Universal Robots PolyScope program: pallet_126.urp

Program pallet_126 (createdIn=3.2.19293 lastSavedIn=3.2.19293 directory=/programs installation=default robotSerialNumber=2015351391)
Calibrated DH parameters: a=[0.000352, -0.161198, -0.373486, 0.00005, 0.000049, 0]; d=[0.089268, 352.477598, -320.08558, -32.281492, 0.094939, 0.082518]; alpha=[1.570728, 0.001116, -0.003686, 1.571189, -1.570572, 0]; deltaTheta=[-0.000012, 1.181849, -1.491165, 0.309495, -0.000007, 0.000025]
Robot Program (runOnlyOnce=false motionType=MoveJ speed=1.047198 acceleration=1.396263 recalculateMotions=false)
  Pallet pattern(dimensionality=Square firstAxisCount=3 secondAxisCount=3 thirdAxisCount=5 motionType=MoveL speed=0.25 acceleration=1.2 recalculateMotions=false, counterVariable(name=cnt_1, initializeExpression=0), patternPoseVariable(name=位姿_1), feature=Base, children(Waypoint(type=Fixed name=a1st_Corner_1, position(joints=2.5763556957244873, -2.0812442938434046, -2.0229433218585413, -0.5034664312945765, 1.591776967048645, -0.26194888750185186 pose=-0.39287493474301816, 0.3789089223527664, 0.06616154798695834, -2.460791536512403, -1.8027009363597946, 0.090316902258006), poseInFeatureCoordinates=[-0.392875, 0.378909, 0.066162, -2.460792, -1.802701, 0.090317], outputFlangePose=[-0.392865, 0.378909, 0.066161, -2.460798, -1.802654, 0.090216]), Waypoint(type=Fixed name=a2nd_Corner_1, position(joints=2.3224451541900635, -2.320186440144674, -1.5487983862506312, -0.7482627073871058, 1.5784262418746948, -0.5291169325457972 pose=-0.386611770730188, 0.5758943302513561, 0.06650521658612327, -2.446947628948111, -1.8165459438339622, 0.030894912998256457), poseInFeatureCoordinates=[-0.386612, 0.575894, 0.066505, -2.446948, -1.816546, 0.030895], outputFlangePose=[-0.386628, 0.575892, 0.066482, -2.446977, -1.816542, 0.030841]), Waypoint(type=Fixed name=a3rd_Corner_1, position(joints=2.0719354207892664, -2.1626037568261713, -1.8315477023713154, -0.6285018266102558, 1.6020367779501523, -0.7786933796104183 pose=-0.19145307853450216, 0.5759079217417217, 0.07306667136931888, -2.446955511533883, -1.8165637951887514, 0.030572269090385032), poseInFeatureCoordinates=[-0.191453, 0.575908, 0.073067, -2.446956, -1.816564, 0.030572], outputFlangePose=[-0.191468, 0.575892, 0.07306, -2.446977, -1.816542, 0.030841]), Waypoint(type=Fixed name=a4th_Corner_1, position(joints=2.3161087418842667, -1.8639255502475685, -2.380638872250877, -0.3727480295157033, 1.579937380718258, -0.5354962677601893 pose=-0.19147099564377815, 0.37025084098707506, 0.07306665267587242, -2.4469490165306196, -1.8165403427476172, 0.03091275584599603), poseInFeatureCoordinates=[-0.191471, 0.370251, 0.073067, -2.446949, -1.81654, 0.030913], outputFlangePose=[-0.191468, 0.370234, 0.07306, -2.446977, -1.816542, 0.030841]))); actionSequence(name=托盘序列 motionType=MoveL speed=0.25 acceleration=1.2 recalculateMotions=false, anchorWaypoint(type=Fixed name=模式点_1, position(joints=2.5763556957244873, -2.0812442938434046, -2.0229433218585413, -0.5034664312945765, 1.591776967048645, -0.26194888750185186 pose=-0.3928301289060624, 0.37891896691542926, 0.06613063584092518, -2.4609637335403103, -1.8026122600963608, 0.0901348807095232), poseInFeatureCoordinates=[-0.39283, 0.378919, 0.066131, -2.460964, -1.802612, 0.090135], outputFlangePose=[-0.392865, 0.378909, 0.066161, -2.460798, -1.802654, 0.090216]), feature=Base, children(Waypoint(type=Fixed name=方式_1, position(joints=2.5763106641148106, -1.8432385802402793, -1.926417143951463, -0.8379843652254397, 1.5904283279567348, -0.2613920478888616 pose=-0.39285064321590996, 0.3789340637699954, 0.19594684257979098, -2.460839566654045, -1.8025601228199282, 0.09032804072053387), poseInFeatureCoordinates=[-0.392851, 0.378934, 0.195947, -2.46084, -1.80256, 0.090328], outputFlangePose=[-0.392865, 0.378909, 0.19594, -2.460798, -1.802654, 0.090216]), Waypoint=模式点_1, Set(type=DigitalOutput, pin=Lamp, digitalValue=1), Wait(type=Sleep, waitTime=1), Waypoint(type=Fixed name=退出_1, position(joints=2.5763106641148106, -1.8432385802402793, -1.926417143951463, -0.8379843652254397, 1.5904283279567348, -0.2613920478888616 pose=-0.3928538096165732, 0.3789354788600276, 0.19593739894347656, -2.4607717536330296, -1.8026458385217325, 0.0899629353725573), poseInFeatureCoordinates=[-0.392854, 0.378935, 0.195937, -2.460772, -1.802646, 0.089963], outputFlangePose=[-0.392865, 0.378909, 0.19594, -2.460798, -1.802654, 0.090216])))
    Pattern -> pattern
    AnchoredSequence -> 托盘序列
